Yaskawa INFORM job: SKRZYNIA_5040_180_STOPNI_30BR.JBI

/JOB
//NAME SKRZYNIA_5040_180_STOPNI_30BR
///FOLDERNAME 02-SKRZYNIE_JOBS
//POS
///NPOS 314,314,0,19,0,0
///TOOL 0
///POSTYPE PULSE
///PULSE
C00000=0,-52280,40443,0,6876,0
C00001=22046,-37966,39112,130493,-19155,27174
C00002=84284,-61498,-6635,149088,14842,16513
C00003=84338,-61498,-27685,149088,14842,16513
C00004=82698,-50112,-46350,149088,16213,11860
C00005=39892,-32884,-45211,76150,37463,9037
C00006=29578,-17223,-58449,88744,50523,9238
C00007=35972,-17118,-57253,86400,42961,7508
C00008=35458,-15932,-56221,86377,43275,7627
C00009=34480,-13589,-54127,86364,43873,7834
C00010=36072,-13496,-54043,85834,42913,7858
C00011=35458,-15932,-56221,86377,43275,7627
C00012=35972,-17118,-57253,86400,42961,7508
C00013=36651,-18645,-58554,86449,42543,7341
C00014=40131,-33875,-57906,55787,43018,13229
C00015=42877,-27397,-54480,52073,42944,15327
C00016=41279,-24645,-52415,52489,44168,15270
C00017=43050,-24404,-52230,51392,43274,15749
C00018=42877,-27397,-54480,52073,42944,15327
C00019=40898,-20830,-25780,49157,48098,14521
C00020=62318,32,1961,9986,53101,20710
C00021=57232,-2732,-5702,17854,51831,19886
C00022=55908,-874,-3716,18514,52152,19396
C00023=57251,-361,-3163,17839,51861,19902
C00024=57232,-2732,-5702,17854,51831,19886
C00025=38366,-25228,-29715,60491,44767,12858
C00026=72952,-57726,-43284,78667,23091,3368
C00027=83918,-61953,-48743,149551,29621,-25735
C00028=40577,-31455,-39147,101508,36831,1521
C00029=54617,-27930,-62814,115696,20453,2389
C00030=55104,-21653,-58012,112587,19523,3879
C00031=52639,-18308,-55249,110097,20657,5472
C00032=54107,-17941,-54938,110495,19799,5062
C00033=54054,-22496,-58686,112518,20186,4058
C00034=53559,-27993,-62861,115181,21045,2810
C00035=46424,-32589,-51504,107545,30005,2440
C00036=40681,-36168,-63553,67140,38442,15724
C00037=40681,-33941,-43766,82094,35701,6883
C00038=41605,-28734,-40246,79922,35248,8110
C00039=39594,-25457,-37847,79253,36712,8594
C00040=41971,-24989,-37494,78590,35137,8865
C00041=41605,-28734,-40246,79922,35248,8110
C00042=39595,-34264,-43971,82374,36430,6754
C00043=39595,-34264,-43971,82374,36430,6754
C00044=60675,5104,-1198,11697,63109,20495
C00045=58712,7984,2210,12440,63222,19806
C00046=59959,8614,2971,11986,62991,20226
C00047=60675,5104,-1198,11697,63109,20495
C00048=54921,-25705,-45327,20944,49629,23906
C00049=89861,-79075,-64611,123776,2144,-16352
C00050=90185,-75920,-61074,-32632,-3931,57195
C00051=86028,-64310,-60026,34123,6588,25352
C00052=40577,-31455,-39147,101508,36831,1521
C00053=43444,-31174,-39127,109807,34843,-777
C00054=44411,-26257,-38426,105777,33065,1485
C00055=42583,-23438,-36280,104470,34034,2315
C00056=44206,-23266,-36146,104768,32979,2063
C00057=44411,-26257,-38426,105777,33065,1485
C00058=41368,-34890,-44347,108169,35847,229
C00059=40577,-31455,-39147,101508,36831,1521
C00060=40577,-27956,-24714,110033,39226,-3600
C00061=43354,-28377,-30152,60321,36920,10063
C00062=43938,-23149,-26293,58645,37185,11059
C00063=42339,-20723,-24375,58783,38386,10986
C00064=44226,-20417,-24125,57897,37300,11501
C00065=43938,-23149,-26293,58645,37185,11059
C00066=40577,-31455,-39147,101508,36831,1521
C00067=86028,-64310,-60026,34123,6588,25352
C00068=86028,-64310,-60026,57978,24772,25352
C00069=86028,-64309,-60028,57978,24769,25352
C00070=40577,-31455,-39147,101508,36831,1521
C00071=40577,-31455,-39147,101508,36831,1521
C00072=38004,-8862,-6434,128891,58396,-6841
C00073=38416,-3307,-839,128870,57964,-6812
C00074=37262,-678,1960,128510,58508,-6504
C00075=38358,-729,1907,128831,57958,-6778
C00076=38416,-3307,-839,128870,57964,-6812
C00077=38733,-19354,-20733,114988,46978,-4200
C00078=41982,-30471,-41162,75746,36694,8784
C00079=73009,-40277,-6382,95546,11240,-8083
C00080=45844,-59376,-6382,28358,16063,-8083
C00081=0,-52280,40443,0,6876,0
C00082=0,-52280,40443,0,6876,0
C00083=-1604,-53109,36209,-13408,3610,-1485
C00084=-84284,-61498,-6635,-149088,14842,-16513
C00085=-84338,-61498,-27685,-149088,14842,-16513
C00086=-82698,-50112,-46350,-149088,16213,-11860
C00087=-39926,-32871,-45210,-76130,37442,-9048
C00088=-29605,-17209,-58453,-88725,50507,-9245
C00089=-35997,-17103,-57256,-86378,42945,-7517
C00090=-36161,-15590,-55863,-86139,42849,-7639
C00091=-35398,-13811,-54272,-86136,43316,-7796
C00092=-37060,-13663,-54140,-85569,42316,-7827
C00093=-36161,-15590,-55863,-86139,42849,-7639
C00094=-35997,-17103,-57256,-86378,42945,-7517
C00095=-36677,-18629,-58556,-86426,42527,-7351
C00096=-40166,-33858,-57895,-55763,43001,-13241
C00097=-44106,-26709,-53973,-51185,42404,-15742
C00098=-42813,-24563,-52349,-51561,43374,-15671
C00099=-44066,-24591,-52370,-50799,42721,-15997
C00100=-44106,-26709,-53973,-51185,42404,-15742
C00101=-40870,-31947,-42232,-63836,39356,-11267
C00102=-59567,-18910,-30925,-15623,47173,-21537
C00103=-46326,-23755,-35701,-49047,38797,-12459
C00104=-45215,-22112,-34410,-49381,39603,-12311
C00105=-46873,-21854,-34207,-48350,38771,-12857
C00106=-46326,-23755,-35701,-49047,38797,-12459
C00107=-40577,-31455,-39147,-101508,36831,-1521
C00108=-83918,-61953,-48743,-149551,29621,25735
C00109=-83918,-61953,-48743,-149551,29621,25735
C00110=-40577,-31455,-39147,-101508,36831,-1521
C00111=-54617,-27930,-62814,-115696,20453,-2389
C00112=-56579,-20436,-56910,-112918,18628,-3510
C00113=-54441,-17635,-54560,-110690,19618,-4917
C00114=-55807,-17308,-54280,-111137,18824,-4501
C00115=-56579,-20436,-56910,-112918,18628,-3510
C00116=-53559,-27993,-62861,-115181,21045,-2810
C00117=-46424,-32589,-51504,-107545,30005,-2440
C00118=-40681,-36168,-63553,-67140,38442,-15724
C00119=-48096,-30599,-43096,-42650,39511,-17645
C00120=-50542,-24010,-38286,-39708,39613,-19319
C00121=-48645,-21434,-36253,-40588,40865,-18895
C00122=-50201,-21153,-36025,-39495,40213,-19474
C00123=-50542,-24010,-38286,-39708,39613,-19319
C00124=-47108,-31001,-43369,-43375,39900,-17247
C00125=-42092,-32720,-44065,-59648,38266,-12707
C00126=-44478,-28697,-29800,-58406,35076,-10579
C00127=-48490,-26278,-44323,-32151,49147,-14295
C00128=-38294,-11895,-19478,-43175,56952,-10784
C00129=-43474,-9694,-17319,-41165,54649,-12265
C00130=-41958,-6845,-14529,-41653,55511,-11926
C00131=-43433,-6608,-14293,-41072,54841,-12342
C00132=-43474,-9694,-17319,-41165,54649,-12265
C00133=-40345,-33419,-45947,-59645,39680,-12787
C00134=-86028,-64310,-60024,-34123,6590,-25350
C00135=-86028,-64310,-60026,-34123,6588,-25352
C00136=-86028,-64310,-60026,-34123,6588,-25352
C00137=-40577,-31455,-39147,-101508,36831,-1521
C00138=-43444,-31174,-39127,-109807,34843,777
C00139=-46521,-24543,-34262,-108607,32275,188
C00140=-44940,-22248,-32476,-107418,33095,-535
C00141=-46605,-21996,-32278,-107847,32021,-235
C00142=-46521,-24543,-34262,-108607,32275,188
C00143=-41368,-34890,-44347,-108169,35847,-229
C00144=-40577,-31455,-39147,-101508,36831,-1521
C00145=-40577,-27956,-24714,-110033,39226,3600
C00146=-43354,-28377,-30152,-60321,36920,-10063
C00147=-46756,-22511,-26749,-56446,35933,-12334
C00148=-45024,-20038,-24770,-56735,37201,-12185
C00149=-46449,-19924,-24676,-56017,36388,-12591
C00150=-46756,-22511,-26749,-56446,35933,-12334
C00151=-40577,-31455,-39147,-101508,36831,-1521
C00152=-86028,-64310,-60026,-34123,6588,-25352
C00153=-86028,-64310,-60026,-57978,24772,-25352
C00154=-59143,-71667,-51735,-34693,44119,-20682
C00155=0,-52280,40443,0,6876,0
C00156=0,-52280,40443,0,6876,0
C00157=15812,-52280,40443,0,6876,0
C00158=17840,-61498,-6635,149088,-29435,16513
C00159=84284,-61498,-6635,149088,14842,16513
C00160=84338,-61498,-27685,149088,14842,16513
C00161=82698,-50112,-46350,149088,16213,11860
C00162=39892,-32884,-45211,76150,37463,9037
C00163=29578,-17223,-58449,88744,50523,9238
C00164=35972,-17118,-57253,86400,42961,7508
C00165=35462,-16432,-53552,88622,43277,6159
C00166=35771,-13988,-51380,88183,43081,6386
C00167=35862,-12801,-56410,83681,43133,9302
C00168=35462,-16432,-53552,88622,43277,6159
C00169=35972,-17118,-57253,86400,42961,7508
C00170=36651,-18645,-58554,86449,42543,7341
C00171=40131,-33875,-57906,55787,43018,13229
C00172=42875,-27281,-50306,54501,41341,13772
C00173=42838,-24414,-54207,50440,44212,16406
C00174=42883,-24331,-48080,53872,41725,14170
C00175=42875,-27281,-50306,54501,41341,13772
C00176=38840,-28785,-40054,63699,40977,11434
C00177=60557,-12849,-28397,13500,50606,22264
C00178=60557,-12849,-28397,13500,50606,22264
C00179=59758,-11739,-27367,13975,50861,21975
C00180=54558,-1776,-20452,19413,63710,22921
C00181=57450,-8787,-40303,15298,66374,23814
C00182=40836,-31962,-42240,63856,39375,11256
C00183=82343,-65193,-54527,93610,14032,-4330
C00184=84338,-61498,-27685,149088,14842,16513
C00185=84284,-61498,-6635,149088,14842,16513
C00186=17840,-61498,-6635,149088,-29435,16513
C00187=3723,-43557,57000,-17428,2162,9388
C00188=8378,-45465,40443,0,6876,0
C00189=-13804,-40918,31830,-137803,-19104,-21261
C00190=-84284,-61498,-6635,-149088,14842,-16513
C00191=-84338,-61498,-27685,-149088,14842,-16513
C00192=-82698,-50112,-46350,-149088,16213,-11860
C00193=-39926,-32871,-45210,-76130,37442,-9048
C00194=-29605,-17209,-58453,-88725,50507,-9245
C00195=-35997,-17103,-57256,-86378,42945,-7517
C00196=-35488,-16417,-53555,-88601,43261,-6168
C00197=-36745,-14323,-51699,-87946,42480,-6360
C00198=-36749,-13075,-56679,-83369,42608,-9309
C00199=-35488,-16417,-53555,-88601,43261,-6168
C00200=-35997,-17103,-57256,-86378,42945,-7517
C00201=-36677,-18629,-58556,-86426,42527,-7351
C00202=-40166,-33858,-57895,-55763,43001,-13241
C00203=-42907,-27264,-50294,-54478,41326,-13783
C00204=-43848,-24488,-54264,-49825,43692,-16665
C00205=-43781,-24493,-48206,-53380,41218,-14381
C00206=-42907,-27264,-50294,-54478,41326,-13783
C00207=-31488,-23274,-37316,-66071,52131,-11172
C00208=-56300,-17768,-33184,-19067,49227,-20577
C00209=-60622,-11441,-27072,-13431,50739,-22310
C00210=-53579,-2503,-19486,-21788,61784,-22236
C00211=-48017,-10819,-42976,-22029,70972,-22007
C00212=-48017,-10819,-42976,-22029,70972,-22007
C00213=-83918,-61953,-48743,-149551,29621,25735
C00214=-84338,-61498,-27685,-149088,14842,-16513
C00215=-84284,-61498,-6635,-149088,14842,-16513
C00216=-17840,-61498,-6635,-149088,-29435,-16513
C00217=10089,-52280,40443,0,6876,0
C00218=83918,-61953,-48743,149551,29621,-25735
C00219=83918,-61953,-48743,149551,29621,-25735
C00220=40577,-31455,-39147,101508,36831,1521
C00221=54617,-27930,-62814,115696,20453,2389
C00222=55104,-21653,-58012,112587,19523,3879
C00223=53867,-18413,-52210,115604,20932,2535
C00224=53940,-17506,-57605,104897,19115,7878
C00225=54054,-22496,-58686,112518,20186,4058
C00226=53559,-27993,-62861,115181,21045,2810
C00227=46424,-32589,-51504,107545,30005,2440
C00228=48066,-32059,-56324,37139,45577,21196
C00229=48065,-29274,-35956,46116,36788,15559
C00230=48424,-24788,-35779,42982,38883,17426
C00231=48349,-21239,-32999,42408,39464,17779
C00232=48348,-19917,-25689,45960,36632,15643
C00233=48424,-24788,-35779,42982,38883,17426
C00234=47075,-29662,-36224,46826,37219,15157
C00235=100689,-57813,-50408,-28184,14534,53618
C00236=97362,-69922,-53058,-41123,7265,59550
C00237=85591,-71083,-59247,22337,12917,31375
C00238=35517,-7803,3690,121195,57133,-9073
C00239=35165,-715,17920,123161,59944,-10941
C00240=35243,-3902,7611,120988,57147,-8910
C00241=35517,-7803,3690,121195,57133,-9073
C00242=37169,-28868,-19142,95064,49514,-4729
C00243=76155,-51955,-34982,81049,11094,2542
C00244=0,-52280,40443,0,6876,0
C00245=-83918,-61953,-48743,-149551,29621,25735
C00246=-40577,-31455,-39147,-101508,36831,-1521
C00247=-54617,-27930,-62814,-115696,20453,-2389
C00248=-55104,-21653,-58012,-112587,19523,-3879
C00249=-55687,-17880,-51757,-116402,19892,-1896
C00250=-55676,-16677,-56890,-104952,18070,-7597
C00251=-54054,-22496,-58686,-112518,20186,-4058
C00252=-53559,-27993,-62861,-115181,21045,-2810
C00253=-46424,-32589,-51504,-107545,30005,-2440
C00254=-51041,-28525,-71952,-25943,59083,-26409
C00255=-51039,-30177,-54804,-30457,47642,-22792
C00256=-51185,-24567,-53701,-28900,50583,-23908
C00257=-52395,-20409,-50395,-27776,50948,-24555
C00258=-52358,-20578,-44444,-29523,47279,-23285
C00259=-51185,-24567,-53701,-28900,50583,-23908
C00260=-50092,-30635,-55121,-31144,47866,-22425
C00261=-97134,-60592,-70548,10988,29316,-44040
C00262=-97134,-60592,-70548,10988,29316,-44040
C00263=-35646,-23010,-11792,-87952,46459,3318
C00264=-30761,-10321,-10113,-87397,53231,-206
C00265=-30869,-8269,-1615,-90458,53281,2257
C00266=-28670,-14621,-14060,-87724,54661,85
C00267=-33867,-15621,4670,-92735,45427,5524
C00268=-86028,-64310,-60024,-34123,6590,-25350
C00269=-52835,-59760,-20413,-18729,6532,-16470
C00270=0,-52280,40443,0,6876,0
C00271=86028,-64310,-60026,34123,6588,25352
C00272=86028,-64310,-60026,34123,6588,25352
C00273=40577,-31455,-39147,101508,36831,1521
C00274=43444,-31174,-39127,109807,34843,-777
C00275=44411,-24891,-31035,111214,34582,-1606
C00276=43990,-22048,-28837,110265,34587,-1050
C00277=43982,-23361,-36098,104874,33158,2017
C00278=44411,-24891,-31035,111214,34582,-1606
C00279=41368,-34890,-44347,108169,35847,229
C00280=40577,-31455,-39147,101508,36831,1521
C00281=40577,-27956,-24714,110033,39226,-3600
C00282=43354,-28377,-30152,60321,36920,10063
C00283=43938,-23847,-29499,56832,38038,12143
C00284=43904,-21311,-27511,56288,38341,12475
C00285=43921,-19578,-19753,60716,36328,9839
C00286=43938,-23847,-29499,56832,38038,12143
C00287=40577,-31455,-39147,101508,36831,1521
C00288=86028,-64310,-60026,34123,6588,25352
C00289=86028,-64310,-60026,57978,24772,25352
C00290=76655,-63519,-28491,15472,11851,31836
C00291=0,-52280,40443,0,6876,0
C00292=0,-52280,40443,0,6876,0
C00293=-86028,-64310,-60026,-34123,6588,-25352
C00294=-86028,-64310,-60026,-34123,6588,-25352
C00295=-40577,-31455,-39147,-101508,36831,-1521
C00296=-43444,-31174,-39127,-109807,34843,777
C00297=-44411,-24891,-31035,-111214,34582,1606
C00298=-46306,-21354,-28285,-110909,33087,1469
C00299=-46340,-22527,-35442,-105171,31587,-1734
C00300=-44411,-24891,-31035,-111214,34582,1606
C00301=-41368,-34890,-44347,-108169,35847,-229
C00302=-40577,-31455,-39147,-101508,36831,-1521
C00303=-40577,-27956,-24714,-110033,39226,3600
C00304=-43354,-28377,-30152,-60321,36920,-10063
C00305=-43938,-23847,-29499,-56832,38038,-12143
C00306=-46071,-20446,-26814,-55040,37186,-13174
C00307=-46151,-18893,-19188,-59636,35040,-10486
C00308=-43938,-23847,-29499,-56832,38038,-12143
C00309=-40577,-31455,-39147,-101508,36831,-1521
C00310=-86028,-64310,-60026,-34123,6588,-25352
C00311=-86028,-64310,-60026,-57978,24772,-25352
C00312=-45844,-59376,-6382,-28358,16063,8083
C00313=0,-52280,40443,0,6876,0
BC00000=507149
BC00001=467540
BC00002=467540
BC00003=467540
BC00004=476695
BC00005=477973
BC00006=477973
BC00007=477973
BC00008=477973
BC00009=477973
BC00010=477973
BC00011=477973
BC00012=477973
BC00013=477973
BC00014=477973
BC00015=477970
BC00016=477970
BC00017=477970
BC00018=477970
BC00019=439571
BC00020=439569
BC00021=454932
BC00022=454932
BC00023=454932
BC00024=454932
BC00025=454932
BC00026=454932
BC00027=675626
BC00028=675626
BC00029=700495
BC00030=700495
BC00031=700495
BC00032=700495
BC00033=700495
BC00034=700493
BC00035=686402
BC00036=686402
BC00037=686402
BC00038=686402
BC00039=686402
BC00040=686402
BC00041=686402
BC00042=686402
BC00043=649890
BC00044=655680
BC00045=655680
BC00046=655680
BC00047=655680
BC00048=626666
BC00049=632763
BC00050=698937
BC00051=849627
BC00052=849627
BC00053=849627
BC00054=849627
BC00055=849627
BC00056=849627
BC00057=849627
BC00058=849627
BC00059=849627
BC00060=849627
BC00061=849627
BC00062=849627
BC00063=849627
BC00064=849627
BC00065=849627
BC00066=849627
BC00067=849627
BC00068=849627
BC00069=1007134
BC00070=1003070
BC00071=1002378
BC00072=1002377
BC00073=1002377
BC00074=1002377
BC00075=1002377
BC00076=1002377
BC00077=1002377
BC00078=1002378
BC00079=965704
BC00080=879640
BC00081=828403
BC00082=757004
BC00083=730971
BC00084=467540
BC00085=467540
BC00086=507176
BC00087=477973
BC00088=477973
BC00089=477973
BC00090=477973
BC00091=477973
BC00092=477973
BC00093=477973
BC00094=477973
BC00095=477973
BC00096=477973
BC00097=477970
BC00098=477970
BC00099=477970
BC00100=477970
BC00101=477973
BC00102=477971
BC00103=516375
BC00104=516375
BC00105=516375
BC00106=516375
BC00107=516375
BC00108=516375
BC00109=675626
BC00110=675626
BC00111=700495
BC00112=700495
BC00113=700495
BC00114=700495
BC00115=700495
BC00116=700493
BC00117=686402
BC00118=686402
BC00119=648000
BC00120=648000
BC00121=648000
BC00122=648000
BC00123=648000
BC00124=648000
BC00125=686402
BC00126=686402
BC00127=686402
BC00128=686402
BC00129=686402
BC00130=686402
BC00131=686402
BC00132=686402
BC00133=651296
BC00134=640664
BC00135=817027
BC00136=849627
BC00137=849627
BC00138=849627
BC00139=849627
BC00140=849627
BC00141=849627
BC00142=849627
BC00143=849627
BC00144=849627
BC00145=849627
BC00146=849627
BC00147=849627
BC00148=849627
BC00149=849627
BC00150=849627
BC00151=849627
BC00152=849627
BC00153=849627
BC00154=842994
BC00155=828403
BC00156=664183
BC00157=467540
BC00158=467540
BC00159=467540
BC00160=467540
BC00161=507176
BC00162=477973
BC00163=477973
BC00164=477973
BC00165=477975
BC00166=477975
BC00167=477975
BC00168=477975
BC00169=477973
BC00170=477973
BC00171=477973
BC00172=477970
BC00173=477970
BC00174=477970
BC00175=477970
BC00176=477973
BC00177=477973
BC00178=477973
BC00179=477973
BC00180=477973
BC00181=461836
BC00182=477973
BC00183=477973
BC00184=467540
BC00185=467540
BC00186=491501
BC00187=513180
BC00188=503726
BC00189=467540
BC00190=467540
BC00191=467540
BC00192=496907
BC00193=477973
BC00194=477973
BC00195=477973
BC00196=477975
BC00197=477975
BC00198=477975
BC00199=477975
BC00200=477973
BC00201=477973
BC00202=477973
BC00203=477970
BC00204=477970
BC00205=477970
BC00206=477970
BC00207=477973
BC00208=477973
BC00209=477973
BC00210=477973
BC00211=477973
BC00212=444232
BC00213=516375
BC00214=467540
BC00215=467540
BC00216=489545
BC00217=503563
BC00218=646286
BC00219=675626
BC00220=675626
BC00221=700495
BC00222=700495
BC00223=700495
BC00224=700495
BC00225=700495
BC00226=700493
BC00227=686402
BC00228=640319
BC00229=640319
BC00230=640319
BC00231=640319
BC00232=640319
BC00233=640319
BC00234=640319
BC00235=605248
BC00236=605248
BC00237=791145
BC00238=763207
BC00239=763207
BC00240=763207
BC00241=763207
BC00242=763207
BC00243=698893
BC00244=541670
BC00245=675626
BC00246=675626
BC00247=700495
BC00248=700495
BC00249=700495
BC00250=700494
BC00251=700495
BC00252=700493
BC00253=686402
BC00254=655680
BC00255=655680
BC00256=655680
BC00257=655680
BC00258=655680
BC00259=655680
BC00260=655680
BC00261=655680
BC00262=769427
BC00263=740449
BC00264=732485
BC00265=732485
BC00266=732485
BC00267=732485
BC00268=780371
BC00269=699504
BC00270=695535
BC00271=817027
BC00272=849627
BC00273=849627
BC00274=849627
BC00275=849627
BC00276=849627
BC00277=849627
BC00278=849627
BC00279=849627
BC00280=849627
BC00281=849627
BC00282=849627
BC00283=849627
BC00284=849627
BC00285=849627
BC00286=849627
BC00287=849627
BC00288=849627
BC00289=849627
BC00290=782138
BC00291=780970
BC00292=695535
BC00293=817027
BC00294=849627
BC00295=849627
BC00296=849627
BC00297=849627
BC00298=849627
BC00299=849627
BC00300=849627
BC00301=849627
BC00302=849627
BC00303=849627
BC00304=849627
BC00305=849627
BC00306=849627
BC00307=849627
BC00308=849627
BC00309=849627
BC00310=849627
BC00311=849627
BC00312=780699
BC00313=789935
///POSTYPE BASE
///RECTAN
///RCONF 0,0,0,0,0,0,0,0,0,0,0,0,0,0,0,0,0,0,0,0,0,0,0,0
P00006=-2.449,0.031,8.825,0.0000,0.0000,0.0000
P00056=0.000,0.000,5.000,0.0000,0.0000,0.0000
///RCONF 1,0,0,0,0,0,0,0,0,0,0,0,0,0,0,0,0,0,0,0,0,0,0,0
P00300=-0.036,-1.505,2.318,0.0000,0.0000,0.0000
///RCONF 0,0,0,0,0,0,0,0,0,0,0,0,0,0,0,0,0,0,0,0,0,0,0,0
P00301=0.005,-4.708,-4.628,0.0000,0.0000,0.0000
P00302=0.052,-2.937,-4.426,0.0000,0.0000,0.0000
P00303=-0.004,-1.437,-4.584,0.0000,0.0000,0.0000
P00304=0.028,-1.666,-4.234,0.0000,0.0000,0.0000
P00305=-0.003,-1.920,-3.501,0.0000,0.0000,0.0000
P00306=0.015,-2.252,-3.054,0.0000,0.0000,0.0000
P00307=0.019,-2.151,-5.077,0.0000,0.0000,0.0000
P00308=-0.003,-2.092,-4.888,0.0000,0.0000,0.0000
P00350=11.519,-0.008,1.149,0.0000,0.0000,0.0000
P00351=13.563,-0.027,-0.653,0.0000,0.0000,0.0000
P00352=13.252,-0.027,-0.827,0.0000,0.0000,0.0000
P00353=10.971,-0.082,0.776,0.0000,0.0000,0.0000
P00354=-0.024,2.508,-1.824,0.0000,0.0000,0.0000
P00355=-0.001,2.528,-1.131,0.0000,0.0000,0.0000
P00356=-0.034,2.921,-0.262,0.0000,0.0000,0.0000
P00357=0.003,3.386,-0.091,0.0000,0.0000,0.0000
//INST
///DATE 2024/05/15 09:14
///ATTR SC,RW
///GROUP1 RB1,BS1
NOP
CALL JOB:MOVE_INTO_TUNNEL
MOVJ C00000 BC00000 VJ=30.00
MOVJ C00001 BC00001 VJ=30.00
MOVJ C00002 BC00002 VJ=30.00
MOVJ C00003 BC00003 VJ=30.00
MOVJ C00004 BC00004 VJ=20.00
MOVL C00005 BC00005 V=500.0
MOVL C00006 BC00006 V=500.0
MOVL C00007 BC00007 V=500.0
'------------------------
'W29.4
'------------------------
MOVL C00008 BC00008 V=66.7 PL=0
REFP 3 C00009 BC00009
CALL JOB:SEARCH-R1
IMOV P0056 V=23.0 PL=0
SET P0300 P0006
SFTON P0300
REFP 3 C00010 BC00010
CALL JOB:SEARCH-R1
SET P0300 P0006
SFTON P0300
MOVL C00011 BC00011 V=66.7 PL=0
SFTOF
MOVL C00012 BC00012 V=500.0
MOVL C00013 BC00013 V=500.0
'PRZEJAZD
MOVL C00014 BC00014 V=500.0
'------------------------
'W63.7
'------------------------
MOVL C00015 BC00015 V=166.7 PL=0
REFP 3 C00016 BC00016
CALL JOB:SEARCH-R1
IMOV P0056 V=23.0 PL=0
SET P0301 P0006
SFTON P0301
REFP 3 C00017 BC00017
CALL JOB:SEARCH-R1
SET P0301 P0006
SFTON P0301
MOVL C00018 BC00018 V=66.7 PL=0
SFTOF
MOVL C00019 BC00019 V=500.0
MOVL C00020 BC00020 V=500.0
'------------------------
'W63.10
'------------------------
MOVL C00021 BC00021 V=66.7 PL=0
REFP 3 C00022 BC00022
CALL JOB:SEARCH-R1
IMOV P0056 V=23.0 PL=0
SET P0302 P0006
SFTON P0302
REFP 3 C00023 BC00023
CALL JOB:SEARCH-R1
SET P0302 P0006
SFTON P0302
MOVL C00024 BC00024 V=66.7 PL=0
SFTOF
MOVL C00025 BC00025 V=500.0
'PRZEJAZD
MOVL C00026 BC00026 V=500.0
MOVJ C00027 BC00027 VJ=30.00
MOVL C00028 BC00028 V=500.0
MOVL C00029 BC00029 V=500.0
'------------------------
'W63.12
'------------------------
MOVL C00030 BC00030 V=66.7 PL=0
REFP 3 C00031 BC00031
CALL JOB:SEARCH-R1
IMOV P0056 V=23.0 PL=0
SET P0303 P0006
SFTON P0303
REFP 3 C00032 BC00032
CALL JOB:SEARCH-R1
SET P0303 P0006
SFTON P0303
MOVL C00033 BC00033 V=66.7 PL=0
SFTOF
'PRZEJAZD
MOVL C00034 BC00034 V=500.0
MOVL C00035 BC00035 V=500.0
MOVL C00036 BC00036 V=500.0
MOVL C00037 BC00037 V=500.0
'------------------------
'W29.16
'------------------------
MOVL C00038 BC00038 V=66.7 PL=0
REFP 3 C00039 BC00039
CALL JOB:SEARCH-R1
IMOV P0056 V=23.0 PL=0
SET P0304 P0006
SFTON P0304
REFP 3 C00040 BC00040
CALL JOB:SEARCH-R1
SET P0304 P0006
SFTON P0304
MOVL C00041 BC00041 V=66.7 PL=0
SFTOF
'PRZEJAZD
MOVL C00042 BC00042 V=500.0
MOVJ C00043 BC00043 VJ=20.00
GETE D040 P0304 (1)
GETE D041 P0304 (2)
GETE D042 P0304 (3)
SETE P0305 (1) D040
SETE P0305 (2) D041
SETE P0305 (3) D042
COMM '------------------------
COMM 'W29.19
COMM '------------------------
COMM MOVL C00044 BC00044 V=66.7 PL=0
COMM REFP 3 C00045 BC00045
COMM CALL JOB:SEARCH-R1
COMM IMOV P0056 V=23.0 PL=0
COMM SET P0305 P0006
COMM SFTON P0305
COMM REFP 3 C00046 BC00046
COMM CALL JOB:SEARCH-R1
COMM SET P0305 P0006
COMM SFTON P0305
COMM MOVL C00047 BC00047 V=66.7 PL=0
COMM SFTOF
COMM 'PRZEJAZD
MOVJ C00048 BC00048 VJ=20.00
MOVJ C00049 BC00049 VJ=20.00
MOVJ C00050 BC00050 VJ=30.00
MOVJ C00051 BC00051 VJ=30.00
MOVL C00052 BC00052 V=500.0
MOVL C00053 BC00053 V=500.0
'------------------------
'W29.22
'------------------------
MOVL C00054 BC00054 V=66.7 PL=0
REFP 3 C00055 BC00055
CALL JOB:SEARCH-R1
IMOV P0056 V=23.0 PL=0
SET P0306 P0006
SFTON P0306
REFP 3 C00056 BC00056
CALL JOB:SEARCH-R1
SET P0306 P0006
SFTON P0306
MOVL C00057 BC00057 V=66.7 PL=0
SFTOF
'PRZEJAZD
MOVL C00058 BC00058 V=500.0
MOVL C00059 BC00059 V=500.0
MOVL C00060 BC00060 V=500.0
MOVL C00061 BC00061 V=500.0
'------------------------
'W63.25
'------------------------
MOVL C00062 BC00062 V=66.7 PL=0
REFP 3 C00063 BC00063
CALL JOB:SEARCH-R1
IMOV P0056 V=23.0 PL=0
SET P0307 P0006
SFTON P0307
REFP 3 C00064 BC00064
CALL JOB:SEARCH-R1
SET P0307 P0006
SFTON P0307
MOVL C00065 BC00065 V=66.7 PL=0
SFTOF
'PRZEJAZD
MOVL C00066 BC00066 V=500.0
MOVL C00067 BC00067 V=500.0
MOVL C00068 BC00068 V=500.0
MOVL C00069 BC00069 V=500.0
COMM MOVL C00070 BC00070 V=500.0
COMM MOVL C00071 BC00071 V=500.0
COMM MOVL C00072 BC00072 V=500.0
COMM '------------------------
COMM 'W63.28
COMM '------------------------
COMM MOVL C00073 BC00073 V=66.7 PL=0
COMM REFP 3 C00074 BC00074
COMM CALL JOB:SEARCH-R1
COMM IMOV P0056 V=23.0 PL=0
COMM SET P0308 P0006
COMM SFTON P0308
COMM REFP 3 C00075 BC00075
COMM CALL JOB:SEARCH-R1
COMM SET P0308 P0006
COMM SFTON P0308
COMM MOVL C00076 BC00076 V=66.7 PL=0
COMM SFTOF
COMM MOVL C00077 BC00077 V=500.0
COMM MOVL C00078 BC00078 V=500.0
MOVJ C00079 BC00079 VJ=10.00
MOVJ C00080 BC00080 VJ=30.00
MOVJ C00081 BC00081 VJ=30.00
CALL JOB:FRONT_SEARCH_180ST_5040_1
MOVJ C00082 BC00082 VJ=30.00
MOVJ C00083 BC00083 VJ=50.00
MOVJ C00084 BC00084 VJ=30.00
MOVJ C00085 BC00085 VJ=30.00
MOVJ C00086 BC00086 VJ=30.00
MOVL C00087 BC00087 V=500.0
MOVL C00088 BC00088 V=500.0
MOVL C00089 BC00089 V=500.0
'------------------------
'W29.4
'------------------------
MOVL C00090 BC00090 V=66.7 PL=0
REFP 3 C00091 BC00091
CALL JOB:SEARCH-R1
IMOV P0056 V=23.0 PL=0
SET P0350 P0006
SFTON P0350
REFP 3 C00092 BC00092
CALL JOB:SEARCH-R1
SET P0350 P0006
SFTON P0350
MOVL C00093 BC00093 V=66.7 PL=0
SFTOF
MOVL C00094 BC00094 V=500.0
MOVL C00095 BC00095 V=500.0
'PRZEJAZD
MOVL C00096 BC00096 V=500.0
GETE D040 P0350 (1)
GETE D041 P0350 (2)
GETE D042 P0350 (3)
SETE P0351 (1) D040
SETE P0351 (2) D041
SETE P0351 (3) D042
GETE D040 P0350 (1)
GETE D041 P0350 (2)
GETE D042 P0350 (3)
SETE P0352 (1) D040
SETE P0352 (2) D041
SETE P0352 (3) D042
COMM '------------------------
COMM 'W63.7
COMM '------------------------
COMM MOVL C00097 BC00097 V=66.7 PL=0
COMM REFP 3 C00098 BC00098
COMM CALL JOB:SEARCH-R1
COMM IMOV P0056 V=23.0 PL=0
COMM SET P0351 P0006
COMM SFTON P0351
COMM REFP 3 C00099 BC00099
COMM CALL JOB:SEARCH-R1
COMM SET P0351 P0006
COMM SFTON P0351
COMM MOVL C00100 BC00100 V=66.7 PL=0
COMM SFTOF
COMM MOVL C00101 BC00101 V=500.0
COMM MOVL C00102 BC00102 V=500.0
COMM '------------------------
COMM 'W63.10
COMM '------------------------
COMM MOVL C00103 BC00103 V=66.7 PL=0
COMM REFP 3 C00104 BC00104
COMM CALL JOB:SEARCH-R1
COMM IMOV P0056 V=23.0 PL=0
COMM SET P0352 P0006
COMM SFTON P0352
COMM REFP 3 C00105 BC00105
COMM CALL JOB:SEARCH-R1
COMM SET P0352 P0006
COMM SFTON P0352
COMM MOVL C00106 BC00106 V=66.7 PL=0
COMM SFTOF
COMM MOVL C00107 BC00107 V=500.0
COMM 'PRZEJAZD
MOVL C00108 BC00108 V=500.0
MOVJ C00109 BC00109 VJ=30.00
MOVL C00110 BC00110 V=500.0
MOVL C00111 BC00111 V=500.0
'------------------------
'W63.12
'------------------------
MOVL C00112 BC00112 V=66.7 PL=0
REFP 3 C00113 BC00113
CALL JOB:SEARCH-R1
IMOV P0056 V=23.0 PL=0
SET P0353 P0006
SFTON P0353
REFP 3 C00114 BC00114
CALL JOB:SEARCH-R1
SET P0353 P0006
SFTON P0353
MOVL C00115 BC00115 V=66.7 PL=0
SFTOF
'PRZEJAZD
MOVL C00116 BC00116 V=500.0
MOVL C00117 BC00117 V=500.0
MOVL C00118 BC00118 V=500.0
MOVL C00119 BC00119 V=500.0
'------------------------
'W29.16
'------------------------
MOVL C00120 BC00120 V=66.7 PL=0
REFP 3 C00121 BC00121
CALL JOB:SEARCH-R1
IMOV P0056 V=23.0 PL=0
SET P0354 P0006
SFTON P0354
REFP 3 C00122 BC00122
CALL JOB:SEARCH-R1
SET P0354 P0006
SFTON P0354
MOVL C00123 BC00123 V=66.7 PL=0
SFTOF
GETE D040 P0354 (1)
GETE D041 P0354 (2)
GETE D042 P0354 (3)
SETE P0355 (1) D040
SETE P0355 (2) D041
SETE P0355 (3) D042
COMM 'PRZEJAZD
COMM MOVL C00124 BC00124 V=500.0
COMM MOVL C00125 BC00125 V=500.0
COMM MOVL C00126 BC00126 V=500.0
COMM MOVL C00127 BC00127 V=500.0
COMM MOVL C00128 BC00128 V=500.0
COMM '------------------------
COMM 'W29.19
COMM '------------------------
COMM MOVL C00129 BC00129 V=66.7 PL=0
COMM REFP 3 C00130 BC00130
COMM CALL JOB:SEARCH-R1
COMM IMOV P0056 V=23.0 PL=0
COMM SET P0355 P0006
COMM SFTON P0355
COMM REFP 3 C00131 BC00131
COMM CALL JOB:SEARCH-R1
COMM SET P0355 P0006
COMM SFTON P0355
COMM MOVL C00132 BC00132 V=66.7 PL=0
COMM SFTOF
COMM 'PRZEJAZD
MOVL C00133 BC00133 V=500.0
MOVJ C00134 BC00134 VJ=30.00
MOVJ C00135 BC00135 VJ=30.00
MOVJ C00136 BC00136 VJ=10.00
MOVL C00137 BC00137 V=500.0
MOVL C00138 BC00138 V=500.0
'------------------------
'W29.22
'------------------------
MOVL C00139 BC00139 V=66.7 PL=0
REFP 3 C00140 BC00140
CALL JOB:SEARCH-R1
IMOV P0056 V=23.0 PL=0
SET P0356 P0006
SFTON P0356
REFP 3 C00141 BC00141
CALL JOB:SEARCH-R1
SET P0356 P0006
SFTON P0356
MOVL C00142 BC00142 V=66.7 PL=0
SFTOF
'PRZEJAZD
MOVL C00143 BC00143 V=500.0
MOVL C00144 BC00144 V=500.0
MOVL C00145 BC00145 V=500.0
MOVL C00146 BC00146 V=500.0
'------------------------
'W63.25
'------------------------
MOVL C00147 BC00147 V=66.7 PL=0
REFP 3 C00148 BC00148
CALL JOB:SEARCH-R1
IMOV P0056 V=23.0 PL=0
SET P0357 P0006
SFTON P0357
REFP 3 C00149 BC00149
CALL JOB:SEARCH-R1
SET P0357 P0006
SFTON P0357
MOVL C00150 BC00150 V=66.7 PL=0
SFTOF
'PRZEJAZD
MOVL C00151 BC00151 V=500.0
MOVL C00152 BC00152 V=500.0
MOVL C00153 BC00153 V=500.0
MOVJ C00154 BC00154 VJ=30.00
MOVJ C00155 BC00155 VJ=30.00
MOVJ C00156 BC00156 VJ=30.00
MOVJ C00157 BC00157 VJ=30.00
MOVJ C00158 BC00158 VJ=20.00
MOVJ C00159 BC00159 VJ=10.00
MOVJ C00160 BC00160 VJ=10.00
MOVJ C00161 BC00161 VJ=10.00
MOVL C00162 BC00162 V=500.0
MOVL C00163 BC00163 V=500.0
MOVL C00164 BC00164 V=500.0
'------------------------
'W29.4
'------------------------
MOVL C00165 BC00165 V=66.7
SFTON P0300
MOVL C00166 BC00166 V=66.7 PL=0
MACRO1 MJ#(0) ARGF24
ARCON
MOVL C00167 BC00167 V=10.8
ARCOF
SFTOF
MOVL C00168 BC00168 V=66.7
SFTOF
MOVL C00169 BC00169 V=500.0
MOVL C00170 BC00170 V=500.0
'PRZEJAZD
MOVL C00171 BC00171 V=500.0
'------------------------
'W63.7
'------------------------
MOVL C00172 BC00172 V=66.7
SFTON P0301
MOVL C00173 BC00173 V=66.7 PL=0
MACRO1 MJ#(0) ARGF24
ARCON
MOVL C00174 BC00174 V=10.0
ARCOF
SFTOF
MOVL C00175 BC00175 V=66.7
SFTOF
MOVL C00176 BC00176 V=500.0
MOVL C00177 BC00177 V=500.0
'------------------------
'W63.10
'------------------------
MOVL C00178 BC00178 V=66.7
SFTON P0302
MOVL C00179 BC00179 V=66.7 PL=0
MACRO1 MJ#(0) ARGF24
ARCON
MOVL C00180 BC00180 V=10.8
ARCOF
SFTOF
MOVL C00181 BC00181 V=250.0
SFTOF
MOVL C00182 BC00182 V=500.0
'PRZEJAZD
MOVL C00183 BC00183 V=500.0
MOVJ C00184 BC00184 VJ=10.00
MOVJ C00185 BC00185 VJ=10.00
MOVJ C00186 BC00186 VJ=25.00
MOVJ C00187 BC00187 VJ=25.00
'TEST
'TEST
'TEST
'TEST
MOVJ C00188 BC00188 VJ=20.00
MOVJ C00189 BC00189 VJ=20.00
MOVJ C00190 BC00190 VJ=20.00
MOVJ C00191 BC00191 VJ=20.00
MOVJ C00192 BC00192 VJ=20.00
MOVL C00193 BC00193 V=500.0
MOVL C00194 BC00194 V=500.0
MOVL C00195 BC00195 V=500.0
'------------------------
'W29.4
'------------------------
MOVL C00196 BC00196 V=66.7
SFTON P0350
MOVL C00197 BC00197 V=166.7 PL=0
MACRO1 MJ#(0) ARGF24
ARCON
MOVL C00198 BC00198 V=10.8
ARCOF
SFTOF
MOVL C00199 BC00199 V=250.0
SFTOF
MOVL C00200 BC00200 V=500.0
MOVL C00201 BC00201 V=500.0
'PRZEJAZD
MOVL C00202 BC00202 V=500.0
'------------------------
'W63.7
'------------------------
MOVL C00203 BC00203 V=333.3
SFTON P0351
MOVL C00204 BC00204 V=166.7 PL=0
MACRO1 MJ#(0) ARGF24
ARCON
MOVL C00205 BC00205 V=10.8
ARCOF
SFTOF
MOVL C00206 BC00206 V=166.7
SFTOF
MOVL C00207 BC00207 V=500.0
'------------------------
'W63.10
'------------------------
MOVL C00208 BC00208 V=166.7
SFTON P0352
MOVL C00209 BC00209 V=66.7 PL=0
MACRO1 MJ#(0) ARGF24
ARCON
MOVL C00210 BC00210 V=10.8
ARCOF
SFTOF
MOVL C00211 BC00211 V=166.7
SFTOF
MOVL C00212 BC00212 V=500.0
'PRZEJAZD
MOVL C00213 BC00213 V=500.0
MOVJ C00214 BC00214 VJ=30.00
MOVJ C00215 BC00215 VJ=30.00
MOVJ C00216 BC00216 VJ=30.00
MOVJ C00217 BC00217 VJ=30.00
MOVJ C00218 BC00218 VJ=30.00
MOVJ C00219 BC00219 VJ=10.00
MOVL C00220 BC00220 V=500.0
MOVL C00221 BC00221 V=500.0
'------------------------
'29.13
'------------------------
MOVL C00222 BC00222 V=66.7
SFTON P0303
MOVL C00223 BC00223 V=166.7 PL=0
MACRO1 MJ#(0) ARGF24
ARCON
MOVL C00224 BC00224 V=10.8
ARCOF
SFTOF
MOVL C00225 BC00225 V=250.0
SFTOF
'PRZEJAZD
MOVL C00226 BC00226 V=500.0
MOVL C00227 BC00227 V=500.0
MOVL C00228 BC00228 V=500.0
MOVL C00229 BC00229 V=500.0
'------------------------
'W29.16
'------------------------
MOVL C00230 BC00230 V=250.0
SFTON P0304
MOVL C00231 BC00231 V=166.7 PL=0
MACRO1 MJ#(0) ARGF24
ARCON
MOVL C00232 BC00232 V=10.8
ARCOF
SFTOF
MOVL C00233 BC00233 V=250.0
SFTOF
'PRZEJAZD
MOVL C00234 BC00234 V=500.0
MOVJ C00235 BC00235 VJ=30.00
MOVJ C00236 BC00236 VJ=30.00
MOVJ C00237 BC00237 VJ=20.00
'------------------------
'W29.19
'------------------------
MOVL C00238 BC00238 V=333.3
SFTON P0305
MOVL C00239 BC00239 V=166.7 PL=0
MACRO1 MJ#(0) ARGF24
ARCON
MOVL C00240 BC00240 V=10.8
ARCOF
SFTOF
MOVL C00241 BC00241 V=250.0
SFTOF
'PRZEJAZD
MOVL C00242 BC00242 V=500.0
MOVJ C00243 BC00243 VJ=20.00
MOVJ C00244 BC00244 VJ=30.00
'TEST
'TEST
'TEST
'TEST
MOVJ C00245 BC00245 VJ=10.00
MOVL C00246 BC00246 V=500.0
MOVL C00247 BC00247 V=500.0
'------------------------
'W28.13
'------------------------
MOVL C00248 BC00248 V=166.7
SFTON P0353
MOVL C00249 BC00249 V=166.7 PL=0
MACRO1 MJ#(0) ARGF24
ARCON
MOVL C00250 BC00250 V=10.8
ARCOF
SFTOF
MOVL C00251 BC00251 V=250.0
SFTOF
'PRZEJAZD
MOVL C00252 BC00252 V=500.0
MOVL C00253 BC00253 V=500.0
MOVL C00254 BC00254 V=500.0
MOVL C00255 BC00255 V=500.0
'------------------------
'W28.16
'------------------------
MOVL C00256 BC00256 V=166.7
SFTON P0354
MOVL C00257 BC00257 V=166.7 PL=0
MACRO1 MJ#(0) ARGF24
ARCON
MOVL C00258 BC00258 V=10.8
ARCOF
SFTOF
MOVL C00259 BC00259 V=166.7
SFTOF
'PRZEJAZD
MOVL C00260 BC00260 V=500.0
MOVL C00261 BC00261 V=500.0
MOVJ C00262 BC00262 VJ=30.00
'------------------------
'W28.19
'------------------------
MOVL C00263 BC00263 V=333.3
SFTON P0355
MOVL C00264 BC00264 V=166.7 PL=0
MACRO1 MJ#(0) ARGF24
ARCON
MOVL C00265 BC00265 V=10.8
ARCOF
SFTOF
MOVL C00266 BC00266 V=250.0
SFTOF
'PRZEJAZD
MOVL C00267 BC00267 V=500.0
MOVJ C00268 BC00268 VJ=10.00
MOVJ C00269 BC00269 VJ=30.00
MOVJ C00270 BC00270 VJ=20.00
MOVJ C00271 BC00271 VJ=20.00
MOVJ C00272 BC00272 VJ=20.00
MOVL C00273 BC00273 V=500.0
MOVL C00274 BC00274 V=500.0
'------------------------
'W29.22
'------------------------
MOVL C00275 BC00275 V=66.7
SFTON P0306
MOVL C00276 BC00276 V=166.7 PL=0
MACRO1 MJ#(0) ARGF24
ARCON
MOVL C00277 BC00277 V=10.8
ARCOF
SFTOF
MOVL C00278 BC00278 V=250.0
SFTOF
'PRZEJAZD
MOVL C00279 BC00279 V=500.0
MOVL C00280 BC00280 V=500.0
MOVL C00281 BC00281 V=500.0
MOVL C00282 BC00282 V=500.0
'------------------------
'W63.25
'------------------------
MOVL C00283 BC00283 V=250.0
SFTON P0307
MOVL C00284 BC00284 V=166.7 PL=0
MACRO1 MJ#(0) ARGF24
ARCON
MOVL C00285 BC00285 V=10.8
ARCOF
SFTOF
MOVL C00286 BC00286 V=250.0
SFTOF
'PRZEJAZD
MOVL C00287 BC00287 V=500.0
MOVL C00288 BC00288 V=500.0
MOVL C00289 BC00289 V=500.0
MOVJ C00290 BC00290 VJ=20.00
MOVJ C00291 BC00291 VJ=20.00
'TEST
'TEST
'TEST
MOVJ C00292 BC00292 VJ=20.00
MOVJ C00293 BC00293 VJ=20.00
MOVJ C00294 BC00294 VJ=20.00
MOVL C00295 BC00295 V=500.0
MOVL C00296 BC00296 V=500.0
'------------------------
'W29.22
'------------------------
MOVL C00297 BC00297 V=250.0
SFTON P0356
MOVL C00298 BC00298 V=166.7 PL=0
MACRO1 MJ#(0) ARGF24
ARCON
MOVL C00299 BC00299 V=10.8
ARCOF
SFTOF
MOVL C00300 BC00300 V=250.0
SFTOF
'PRZEJAZD
MOVL C00301 BC00301 V=500.0
MOVL C00302 BC00302 V=500.0
MOVL C00303 BC00303 V=500.0
MOVL C00304 BC00304 V=500.0
'------------------------
'W63.25
'------------------------
MOVL C00305 BC00305 V=66.7
SFTON P0357
MOVL C00306 BC00306 V=166.7 PL=0
MACRO1 MJ#(0) ARGF24
ARCON
MOVL C00307 BC00307 V=10.8
ARCOF
SFTOF
MOVL C00308 BC00308 V=250.0
SFTOF
'PRZEJAZD
MOVL C00309 BC00309 V=500.0
MOVL C00310 BC00310 V=500.0
MOVL C00311 BC00311 V=500.0
MOVJ C00312 BC00312 VJ=30.00
MOVJ C00313 BC00313 VJ=30.00
CALL JOB:FRONT_WELD_180ST_5040_1
CALL JOB:MOVE_OUT_OF_TUNNEL
END
